PROGRAM PRG_07_LineState
VAR
	CheckLine1Producing: CheckLineProducing;
	
	ValueChangeDetector	:	ARRAY[1..6] OF ValueChangeDetector;
	GenericState		:	ARRAY[1..6] OF GenericState;
	PostHttp			:	ARRAY[1..6] OF HttpPost;
	tpValueChangeDelay	:	ARRAY[1..6] OF TP;
	
END_VAR


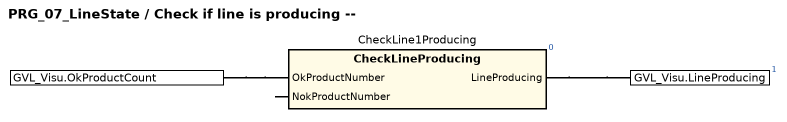
// PAGE Check if line is producing --
CheckLine1Producing(OkProductNumber := GVL_Visu.OkProductCount); // CheckLineProducing
GVL_Visu.LineProducing := CheckLine1Producing.LineProducing;

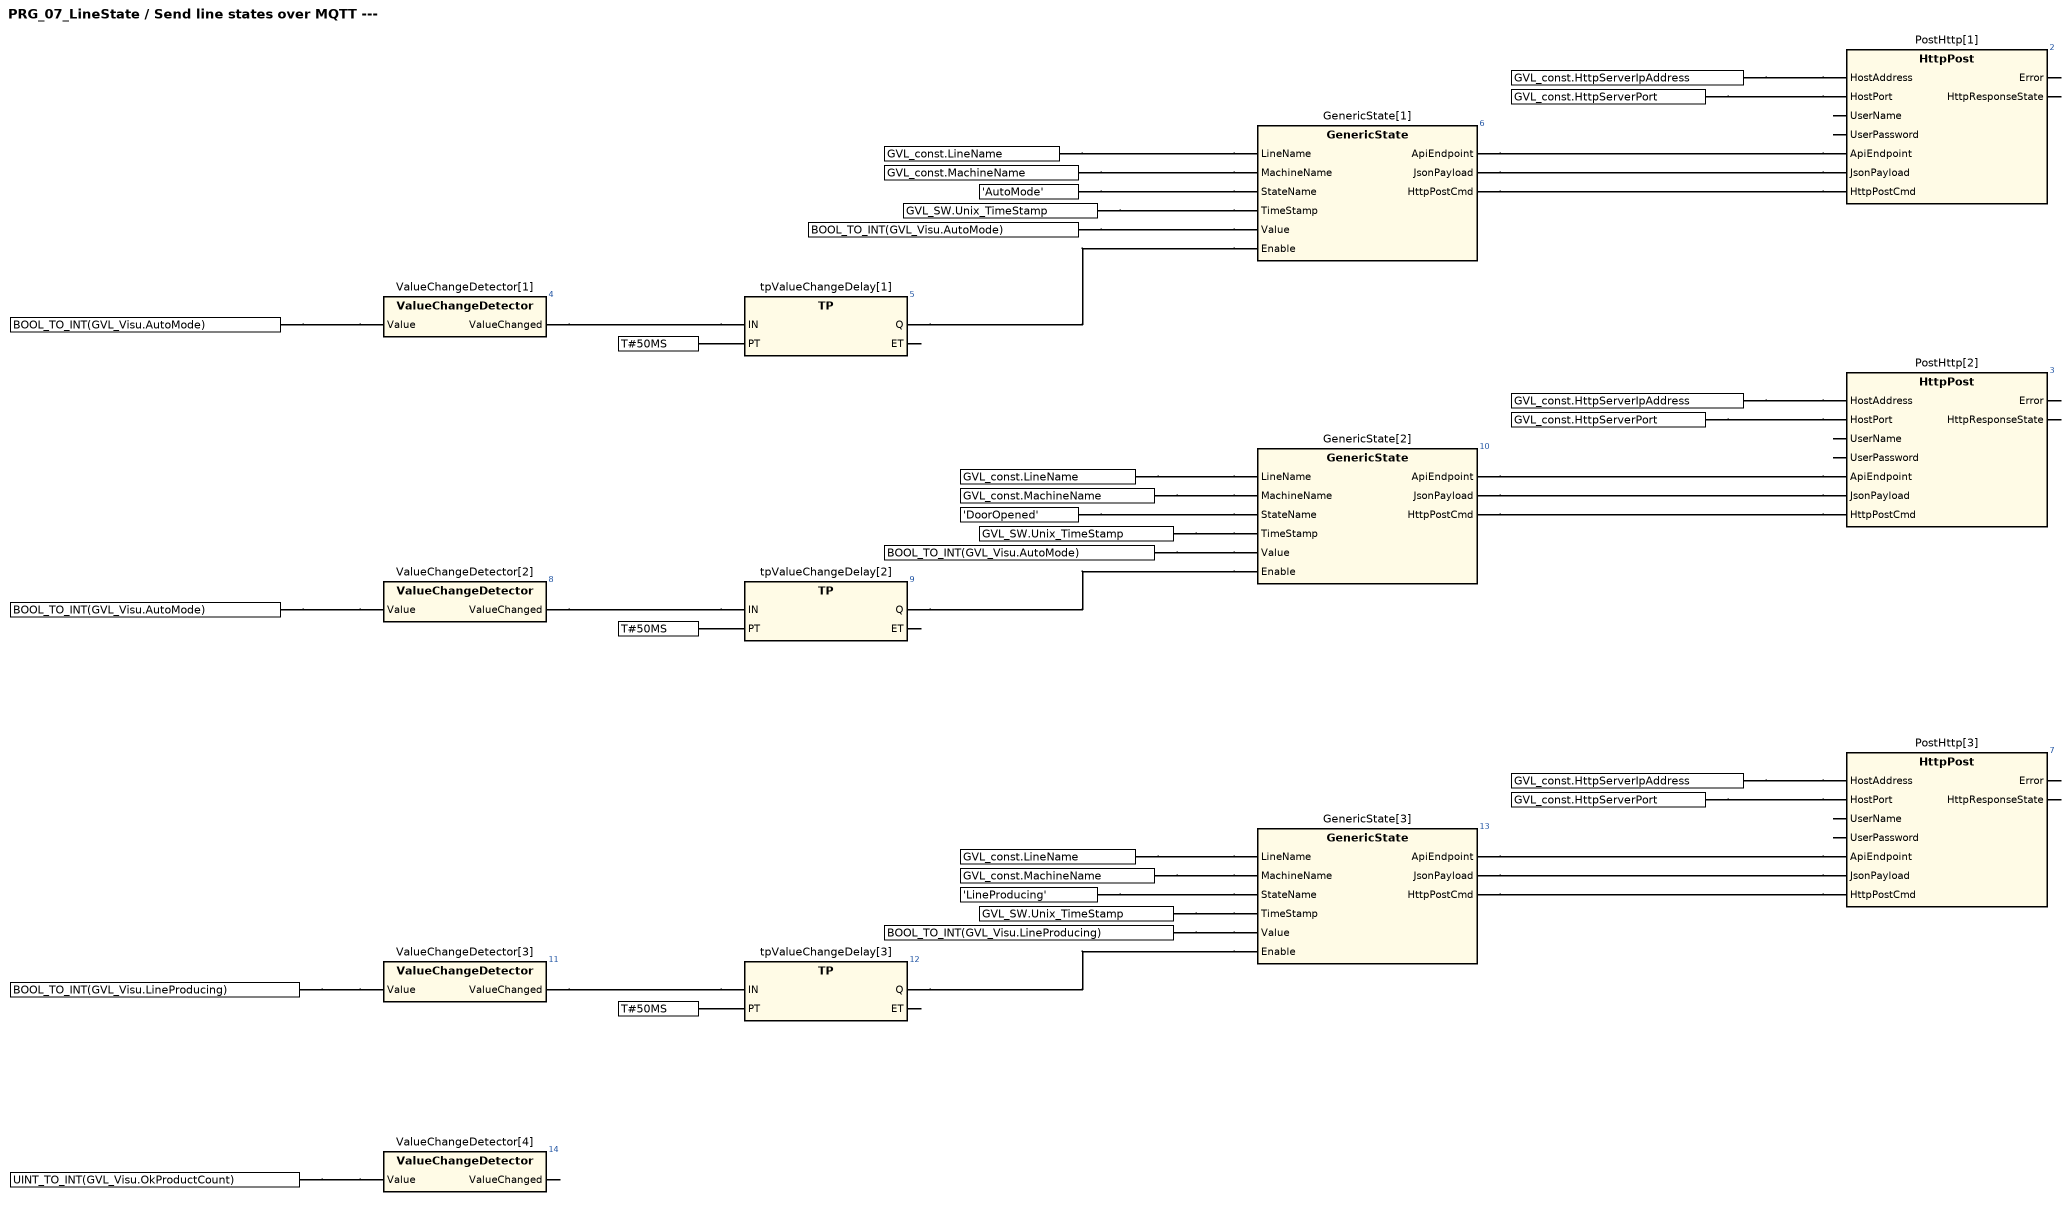
// PAGE Send line states over MQTT ---
PostHttp[1](
    HostAddress := GVL_const.HttpServerIpAddress,
    HostPort := GVL_const.HttpServerPort,
    ApiEndpoint := GenericState[1].ApiEndpoint,
    JsonPayload := GenericState[1].JsonPayload,
    HttpPostCmd := GenericState[1].HttpPostCmd); // HttpPost
PostHttp[2](
    HostAddress := GVL_const.HttpServerIpAddress,
    HostPort := GVL_const.HttpServerPort,
    ApiEndpoint := GenericState[2].ApiEndpoint,
    JsonPayload := GenericState[2].JsonPayload,
    HttpPostCmd := GenericState[2].HttpPostCmd); // HttpPost
ValueChangeDetector[1](Value := BOOL_TO_INT(GVL_Visu.AutoMode)); // ValueChangeDetector
tpValueChangeDelay[1](IN := ValueChangeDetector[1].ValueChanged, PT := T#50MS); // TP
GenericState[1](
    LineName := GVL_const.LineName,
    MachineName := GVL_const.MachineName,
    StateName := 'AutoMode',
    TimeStamp := GVL_SW.Unix_TimeStamp,
    Value := BOOL_TO_INT(GVL_Visu.AutoMode),
    Enable := tpValueChangeDelay[1].Q); // GenericState
PostHttp[3](
    HostAddress := GVL_const.HttpServerIpAddress,
    HostPort := GVL_const.HttpServerPort,
    ApiEndpoint := GenericState[3].ApiEndpoint,
    JsonPayload := GenericState[3].JsonPayload,
    HttpPostCmd := GenericState[3].HttpPostCmd); // HttpPost
ValueChangeDetector[2](Value := BOOL_TO_INT(GVL_Visu.AutoMode)); // ValueChangeDetector
tpValueChangeDelay[2](IN := ValueChangeDetector[2].ValueChanged, PT := T#50MS); // TP
GenericState[2](
    LineName := GVL_const.LineName,
    MachineName := GVL_const.MachineName,
    StateName := 'DoorOpened',
    TimeStamp := GVL_SW.Unix_TimeStamp,
    Value := BOOL_TO_INT(GVL_Visu.AutoMode),
    Enable := tpValueChangeDelay[2].Q); // GenericState
ValueChangeDetector[3](Value := BOOL_TO_INT(GVL_Visu.LineProducing)); // ValueChangeDetector
tpValueChangeDelay[3](IN := ValueChangeDetector[3].ValueChanged, PT := T#50MS); // TP
GenericState[3](
    LineName := GVL_const.LineName,
    MachineName := GVL_const.MachineName,
    StateName := 'LineProducing',
    TimeStamp := GVL_SW.Unix_TimeStamp,
    Value := BOOL_TO_INT(GVL_Visu.LineProducing),
    Enable := tpValueChangeDelay[3].Q); // GenericState
ValueChangeDetector[4](Value := UINT_TO_INT(GVL_Visu.OkProductCount)); // ValueChangeDetector

END_PROGRAM

(* stored: Version 1.1.0.1, ProductVersion 3.1.4024.15
   POU PRG_07_LineState: Id {6b46241e-9a24-414e-99ba-7e1872c65d81}, SpecialFunc None *)
